FUNCTION_BLOCK Test_ListCountIncrements EXTENDS T_UnitTestBase
VAR
    List  : T_ListOfTests(Capacity := 10, TestGroupName := 'Unit Tests');
    Test1 : T_UnitTestBase(List);
END_VAR

Assertion.AssertEquals_DINT(Expected     := 1,
                            Actual       := List.Count,
                            VariableName := 'List.Count');
							
CheckAssertion(NextState := 0);

END_FUNCTION_BLOCK

(* stored: Version 1.1.0.1, ProductVersion 3.1.4024.11
   POU Test_ListCountIncrements: Id {4ad9c475-8d0a-4735-8e26-f4b03d54a0ac}, SpecialFunc None *)
